// TIA Portal V20 export
TYPE "LBP_typeMcp483AdditionalOutput"
TITLE = MCP 483 image / Image du MCP 483
// Additional output image of MCP 483 / Image de sortie supplémentaire du MCP 483
   STRUCT
      reserved1 : Byte;
      optionalKey1 : Bool;   // KT-OUT1,
      optionalKey2 : Bool;   // KT-OUT2
      optionalKey3 : Bool;   // KT-OUT3
      optionalKey4 : Bool;   // KT-OUT4
      optionalKey5 : Bool;   // KT-OUT5
      optionalKey6 : Bool;   // KT-OUT6
      reserved16 : Bool;
      reserved17 : Bool;
   END_STRUCT;
END_TYPE
